(* LS Electric XG5000 project: 05_Practice3_TON_TP *)
(* PLC LSPLC *)
(* module base 0 slot 0: 입력 모듈:XGI-D21A (DC 24V 입력, 8점 (전류소스/싱크입력)) *)
(* module base 0 slot 1: 출력 모듈:XGQ-RY1A (릴레이 출력, 8점 (2A용, 단독 COM.)) *)

PROGRAM NewProgram (* task: 스캔 프로그램 *)
VAR
    물공급타이머 : TP;
    물나옴타이머 : TP;
    세척밸브 AT %QX0.1.0 : BOOL;
    센서 AT %IX0.0.0 : BOOL;
    앉는타이머 : TON;
END_VAR

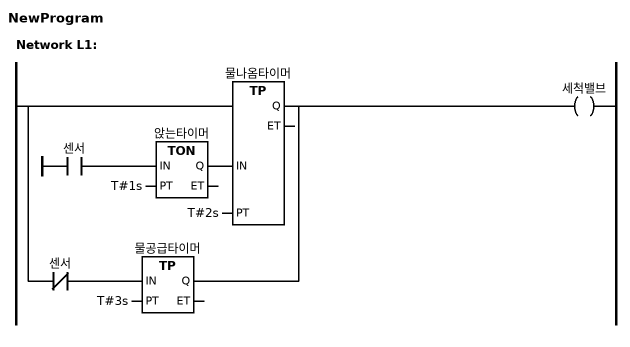
(* Rung L1 *)
앉는타이머(IN := 센서, PT := T#1s);
물나옴타이머(IN := 앉는타이머.Q, PT := T#2s);
물공급타이머(IN := NOT 센서, PT := T#3s);
세척밸브 := 물나옴타이머.Q OR 물공급타이머.Q;
END_PROGRAM